FUNCTION_BLOCK POSTGRES_MEAN_BY_STATION
  {SET_ATTRIBUTE(OpcUa, SERVICE)}
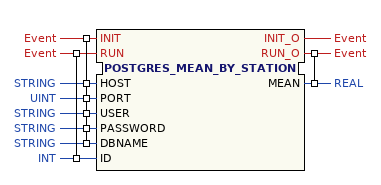
  EVENT_INPUT
    INIT WITH HOST, PORT, USER, PASSWORD, DBNAME;
    RUN WITH ID;
  END_EVENT
  EVENT_OUTPUT
    INIT_O;
    RUN_O WITH MEAN;
  END_EVENT
  VAR_INPUT
    HOST : STRING; {SET_ATTRIBUTE(OpcUa, Constant)}
    PORT : UINT; {SET_ATTRIBUTE(OpcUa, Constant)}
    USER : STRING; {SET_ATTRIBUTE(OpcUa, Constant)}
    PASSWORD : STRING; {SET_ATTRIBUTE(OpcUa, Constant)}
    DBNAME : STRING; {SET_ATTRIBUTE(OpcUa, Constant)}
    ID : INT; {SET_ATTRIBUTE(OpcUa, Constant)}
  END_VAR
  VAR_OUTPUT
    MEAN : REAL; {SET_ATTRIBUTE(OpcUa, Variable)}
  END_VAR
END_FUNCTION_BLOCK
